// TIA Portal V19 export
TYPE "SinamicsCU_Warnings"
// stored: Access Published
   STRUCT
      CUWarning : Bool;   // Warning from CU telegram
      CUSafetyMessagePresence : Bool;   // Safety message presence from CU telegram
   END_STRUCT;
END_TYPE
